Fanuc KAREL source: KF00008.KL

PROGRAM KF00008
%NOLOCKGROUP
VAR
  I: INTEGER
  J: INTEGER
  X: REAL
  Y: REAL
  B: BOOLEAN
  C: BOOLEAN
  TXT: STRING[80]
  TXT2: STRING[80]
  AI: ARRAY[4] OF INTEGER
  BI: ARRAY[4] OF INTEGER
  P: XYZWPR
  JP: JOINTPOS
  PF: POSITION
  V1: VECTOR
  V2: VECTOR
  STATUS: INTEGER
BEGIN
  I = 3
  X = 2.5
  Y = 1.5
  X = X + Y
END KF00008
